// TIA Portal V16 program export: 1 tag tables, 0 data types, 0 data blocks, 1 code blocks (in call order from the OBs), 2 instance data blocks

VAR_GLOBAL   // PLC tag table "Default tag table"
   Y1 AT %Q0.0 : Bool;
   Y2 AT %Q0.1 : Bool;
   H1 AT %Q0.2 : Bool;
   H2 AT %Q0.3 : Bool;
   S1 AT %I0.0 : Bool;
   B1 AT %I0.1 : Bool;
   B2 AT %I0.2 : Bool;
   B3 AT %I0.3 : Bool;
   B4 AT %I0.4 : Bool;
   "Step" AT %MW0 : Int;
END_VAR

ORGANIZATION_BLOCK "Main"   // OB1, LAD, ProgramCycle
TITLE = "Main Program Sweep (Cycle)"
{ S7_Optimized_Access := 'TRUE' }
VERSION : 0.1
// stored: AutoNumber true, IsIECCheckEnabled false, SetENOAutomatically false
   VAR_INPUT
      Initial_Call : Bool;   // Initial call of this OB
      Remanence : Bool;   // =True, if remanent data are available
   END_VAR
   VAR_TEMP   // added for the SCL form of the ladder/FBD networks
      _w1 : Bool;
   END_VAR
BEGIN

REGION Network 1
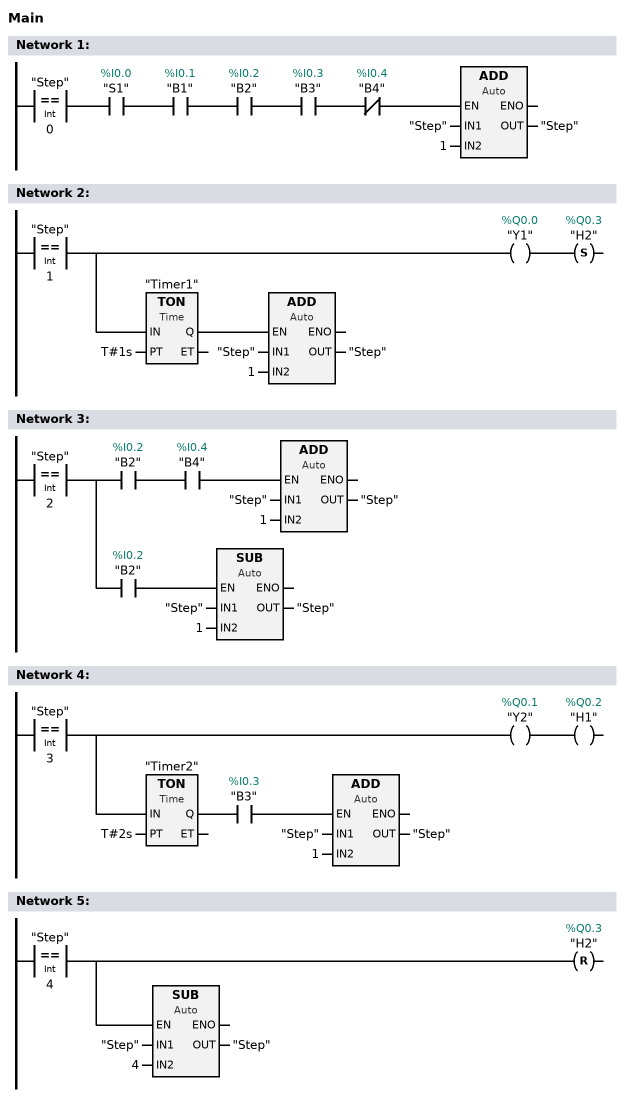
   RUNG wire#powerrail
      { S7_Templates := "SrcType := Int" } EQ_Contact(in1 := "Step", in2 := 0)
      Contact( "S1" )
      Contact( "B1" )
      Contact( "B2" )
      Contact( "B3" )
      I_Contact( "B4" )
      Add(in1 := "Step", in2 := 1, out => "Step")
   END_RUNG
   // the same network as SCL:
   IF ("Step" = 0) AND "S1" AND "B1" AND "B2" AND "B3" AND NOT "B4" THEN "Step" := "Step" + 1; END_IF;
END_REGION

REGION Network 2
   RUNG wire#powerrail
      { S7_Templates := "SrcType := Int" } EQ_Contact(in1 := "Step", in2 := 1)
      wire#w1
      Coil( "Y1" )
      S_Coil( "H2" )
   END_RUNG
   RUNG wire#w1
      { S7_Templates := "time_type := Time" } "Timer1".TON(pt := T#1s, et =>)
      Add(in1 := "Step", in2 := 1, out => "Step")
   END_RUNG
   // the same network as SCL:
   "Y1" := "Step" = 1;
   IF "Y1" THEN "H2" := TRUE; END_IF;
   "Timer1".TON(IN := "Y1", PT := T#1s);
   IF "Timer1".Q THEN "Step" := "Step" + 1; END_IF;
END_REGION

REGION Network 3
   RUNG wire#powerrail
      { S7_Templates := "SrcType := Int" } EQ_Contact(in1 := "Step", in2 := 2)
      wire#w1
      Contact( "B2" )
      Contact( "B4" )
      Add(in1 := "Step", in2 := 1, out => "Step")
   END_RUNG
   RUNG wire#w1
      Contact( "B2" )
      Sub(in1 := "Step", in2 := 1, out => "Step")
   END_RUNG
   // the same network as SCL:
   #_w1 := "Step" = 2;
   IF #_w1 AND "B2" AND "B4" THEN "Step" := "Step" + 1; END_IF;
   IF #_w1 AND "B2" THEN "Step" := "Step" - 1; END_IF;
END_REGION

REGION Network 4
   RUNG wire#powerrail
      { S7_Templates := "SrcType := Int" } EQ_Contact(in1 := "Step", in2 := 3)
      wire#w1
      Coil( "Y2" )
      Coil( "H1" )
   END_RUNG
   RUNG wire#w1
      { S7_Templates := "time_type := Time" } "Timer2".TON(pt := T#2s, et =>)
      Contact( "B3" )
      Add(in1 := "Step", in2 := 1, out => "Step")
   END_RUNG
   // the same network as SCL:
   "Y2" := "Step" = 3;
   "H1" := "Y2";
   "Timer2".TON(IN := "Y2", PT := T#2s);
   IF "Timer2".Q AND "B3" THEN "Step" := "Step" + 1; END_IF;
END_REGION

REGION Network 5
   RUNG wire#powerrail
      { S7_Templates := "SrcType := Int" } EQ_Contact(in1 := "Step", in2 := 4)
      wire#w1
      R_Coil( "H2" )
   END_RUNG
   RUNG wire#w1
      Sub(in1 := "Step", in2 := 4, out => "Step")
   END_RUNG
   // the same network as SCL:
   IF "Step" = 4 THEN
       "H2" := FALSE;
       "Step" := "Step" - 4;
   END_IF;
END_REGION
END_ORGANIZATION_BLOCK

DATA_BLOCK "Timer1"   // DB1
{ S7_Optimized_Access := 'TRUE' }
// stored: AutoNumber true, DBAccessibleFromOPCUA true, InstanceOfName IEC_TIMER, OfSystemLibElement IEC_TIMER, OfSystemLibVersion 1.0
"IEC_TIMER"
   // VAR
   //    PT : Time;
   //    ET { ExternalWritable := 'False'} : Time;
   //    IN : Bool;
   //    Q { ExternalWritable := 'False'} : Bool;
   // END_VAR
BEGIN
END_DATA_BLOCK

DATA_BLOCK "Timer2"   // DB2
{ S7_Optimized_Access := 'TRUE' }
// stored: AutoNumber true, DBAccessibleFromOPCUA true, InstanceOfName IEC_TIMER, OfSystemLibElement IEC_TIMER, OfSystemLibVersion 1.0
"IEC_TIMER"
   // VAR
   //    PT : Time;
   //    ET { ExternalWritable := 'False'} : Time;
   //    IN : Bool;
   //    Q { ExternalWritable := 'False'} : Bool;
   // END_VAR
BEGIN
END_DATA_BLOCK
